PROGRAM PRG_AtTransfer01
VAR
	intnFBSensor : FB_Sensors;
END_VAR

intnFBSensor (
	iSensor := At_Transfer_1,
	iTimeToActuateSensor := 0,
);

END_PROGRAM

(* stored: Version 1.1.0.1
   POU PRG_AtTransfer01: Id {330ff2b7-8217-4ca4-aedc-782079986f95}, SpecialFunc None *)
